# EPICS substitutions: db/Beckhoff_1XXX/ecmcEK1101.substitutions
file "ecmcEcSlave.template"
{
  pattern {}
          {}
}

file "ecmcEK1101-ID.template"
{
  pattern {}
          {}
}
